// TIA Portal V19 export
TYPE "LUC_typeCommands"
TITLE = LUC_typeStateModeManagerCommands
// Module related commands from external systems
// stored: Access Published
   STRUCT
      modeRequests : "LUC_typeModeRequests";   // Commands to request a mode change
      stateCommands : "LUC_typeStateCommands";   // Commands to request a state change
   END_STRUCT;
END_TYPE
